Staubli VAL3: read.pgx

public program read(num pX (dimensions=1), num pY (dimensions=1), string& pMsg[] (dimensions=1), num pLen (dimensions=1), bool pCrypt (dimensions=1))
  local num lLen
  local bool lExit
  local bool lBlk
  local num l
  local num p
  local num lTps
  local string lMsg
  local string lView
  local string lStr
begin
  //---------------------------------
  //  R E A D   O N E   S T R I N G
  //---------------------------------
  // Read one string from the pX
  // column and pY line
  //
  lTps=clock()
  lMsg=pMsg
  p=len(lMsg)
  // cryptage
  if pCrypt
    do
      l=len(lMsg)
      nKey=getKey()
      if ((clock()-lTps)>=0.5)
        if lBlk==true
          lBlk=false
        else
          lBlk=true
        endIf
        lTps=clock()
      endIf
      if (nKey>=32) and (nKey<=126)
        if ((len(lMsg)+1)<=pLen)
          lMsg=lMsg+chr(nKey)
        endIf
      else
        if (nKey==263) and (len(lMsg)>0)
          lMsg=mid(lMsg,len(lMsg)-1,0)
        endIf
      endIf
      if (lStr!=lMsg)
        call strfillchr(lMsg,lView,"*")
        lStr=lMsg
      endIf
      if lBlk==true
        call typeLen(pX,pY,lView+"|",pLen+1)
      else
        call typeLen(pX,pY,lView+" ",pLen+1)
      endIf
      //
      // release the resource
      delay(0)
    until (nKey==270) or (nKey==255)
  else
    // normal read
    // delete the old value
    setTextMode(0)
    call strfillchr(lMsg,lView," ")
    call typeLen(pX,pY,lView,40-pX-1)
    // read the new one
    gotoxy(pX,pY)
    get(lMsg)
  endIf
  // result
  if isKeyPressed(270) or lMsg!=""
    pMsg=lMsg
  endIf
  if isKeyPressed(255)
    bUseEscape=true
  else
    bUseEscape=false
  endIf
end
